// TwinCAT 3 PLC project Test
// ProgramVersion: 3.1.4026.1+c9eadab3edd020c56c333d811d5b3c408c2550c8
// libraries:
//   Tc3_Module, * (Beckhoff Automation GmbH)
//   TcUnit, * (www.tcunit.org)
//   [nepionic-packml], * (nepionic)
// project tree:
//   Mocks/ MockUnitMode.TcPOU
//   Programs/ TestRunner.TcPOU
//   Tasks/ TestRunnerTask.TcTTO
//   Tests/ PackMLTestSuite.TcPOU
// real-time tasks:
//   TASK TestRunnerTask: cycle T#10ms, priority 20, ADS port 350

CONFIGURATION Test
    RESOURCE PLC ON TwinCAT3
        TASK TestRunnerTask(INTERVAL := T#10ms, PRIORITY := 20);
        PROGRAM TestRunner WITH TestRunnerTask : TestRunner;
    END_RESOURCE
END_CONFIGURATION

// ---- Programs/TestRunner.TcPOU
PROGRAM TestRunner
VAR
	packmlTestSuite : PackMLTestSuite;
END_VAR

TcUnit.Run();

END_PROGRAM

// ---- Tests/PackMLTestSuite.TcPOU
FUNCTION_BLOCK PackMLTestSuite EXTENDS TcUnit.FB_TestSuite
VAR
END_VAR

CheckBasicStateMachineCycle();

METHOD PUBLIC CheckBasicStateMachineCycle
VAR
	stateMachine : nepionic_packml.StateMachine;
END_VAR
Test('CheckStateMachine');

AssertTrue(
	Condition := stateMachine.IsIdle,
	Message := 'State machine is not in Idle state immediately after creation'
);

stateMachine.Start();
AssertTrue(
	Condition := stateMachine.IsStarting,
	Message := 'State machine is not in Starting state immediately after Start action'
);

stateMachine.StateComplete();
AssertTrue(
	Condition := stateMachine.IsExecuting,
	Message := 'State machine is not in Execute state immediately after Starting state complete'
);

stateMachine.StateComplete();
AssertTrue(
	Condition := stateMachine.IsCompleting,
	Message := 'State machine is not in Completing state immediately after Execute state complete'
);

stateMachine.StateComplete();
AssertTrue(
	Condition := stateMachine.IsComplete,
	Message := 'State machine is not in Complete state immediately after Completing state complete'
);

stateMachine.Reset();
AssertTrue(
	Condition := stateMachine.IsResetting,
	Message := 'State machine is not in Resetting state immediately after Reset action'
);

stateMachine.StateComplete();
AssertTrue(
	Condition := stateMachine.IsIdle,
	Message := 'State machine is not in Idle state immediately after Resetting state complete'
);

Test_Finished();
END_METHOD

END_FUNCTION_BLOCK

// ---- Mocks/MockUnitMode.TcPOU
{attribute 'linkalways'} 
{attribute 'no_explicit_call' := 'This FB is a CLASS and must be accessed using methods or properties'}
{attribute 'enable_dynamic_creation'}
FUNCTION_BLOCK MockUnitMode EXTENDS nepionic_packml.UnitMode
VAR
END_VAR

END_FUNCTION_BLOCK
